// TIA Portal V15.1 export
// export: Created 2024-05-17T05:38:40.7497504Z, ExportSetting WithDefaults, DisplayName Totally Integrated Automation Portal, DisplayVersion V15.1 Update 5, DisplayName TIA Portal Openness, DisplayVersion V15.1 Update 5, DisplayName SINAMICS Startdrive Advanced, DisplayVersion V15.1, DisplayName G130, G150, S120, S150, SINAMICS MV, S210, DisplayVersion V15.1, DisplayName G110M, G120, G120C, G120D, G120P, DisplayVersion V15.1, DisplayName STEP 7 Professional, DisplayVersion V15.1 Update 5, DisplayName STEP 7 Safety, DisplayVersion V15.1, DisplayName WinCC Professional, DisplayVersion V15.1 Update 5, DisplayName SIMATIC Visualization Architect, DisplayVersion V15.1
FUNCTION "LGBLineFeed-Config" : Void   // FC6643, FBD
TITLE = LGBLineFeed-Config
{ S7_Optimized_Access := 'FALSE' }
AUTHOR : VCC
FAMILY : Control
NAME : Bit2Word
VERSION : 1.0
// stored: AutoNumber false, IsIECCheckEnabled false, SetENOAutomatically False, UDAEnableTagReadback false
   VAR_INPUT
      C_EnableAlarmNoBodyPresent : Bool;   // Enable alarm No Body Present
      C_BodyPitchMinDistance : Bool;   // Body pitch minimum distance is allowed
      C_FixedLineStop_Window : Int;   // Fixed line stop - window where fixed line stop is active (cm)
      C_RampDownDist : Int;   // Ramp down distance of conveyor (cm)
   END_VAR
   VAR_IN_OUT
      IO_Config : "LineFeedConfig";   // Config
   END_VAR
BEGIN

REGION Network 1: **** 1 Inputs **** Config
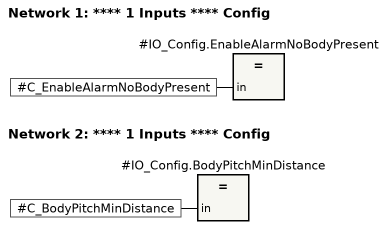
   #IO_Config.EnableAlarmNoBodyPresent := #C_EnableAlarmNoBodyPresent;
END_REGION

REGION Network 2: **** 1 Inputs **** Config
   #IO_Config.BodyPitchMinDistance := #C_BodyPitchMinDistance;
END_REGION

NETWORK
TITLE = **** 1 Inputs **** Move Config UDT
// Move Config
      L     #C_FixedLineStop_Window;
      T     #IO_Config.WindowDist;
      L     #C_RampDownDist;
      T     #IO_Config.RampDownDist;
END_FUNCTION
